// TIA Portal V21 export
TYPE "UDT_Contador"
   STRUCT
      Total : Int;
      Altas : Int;
      Bajas : Int;
   END_STRUCT;
END_TYPE
